FUNCTION Try : BOOL
VAR_INPUT
	iExceptionHandling : I_ExceptionHandling;
END_VAR
VAR_OUTPUT
END_VAR
VAR
END_VAR

END_FUNCTION

(* stored: Version 1.1.0.1, ProductVersion 3.1.4024.0
   POU Try: Id {a5df9670-c639-45b0-bb9d-6f1c178d5eb4}, SpecialFunc None *)
